// TIA Portal V20 export
// export: Created 2025-09-12T17:58:00.0000000Z, ExportSetting WithDefaults
TYPE "UDT500_EM_Monitoring"
   STRUCT
      Dirty_Filter_DI : Bool;   // Digital Input: Dirty filter DP switch (`True` = Dirty).
      Filter_Delay_Sec : Time;   // Time delay for dirty filter alarm (e.g., `T#10s`).
      Dirty_Filter_Alm : Bool;   // Alarm: Dirty filter alarm.
   END_STRUCT;
END_TYPE
